# EPICS autosave request: iocBoot/iocTest/auto_settingsVx.req
file "quadEM_settings.req",            P=$(P), R=QE1:
file "quadEM_TimeSeries_settings.req", P=$(P), R=QE1_TS:
file "quadEM_settings.req",            P=$(P), R=QE2:
file "quadEM_TimeSeries_settings.req", P=$(P), R=QE2_TS:
